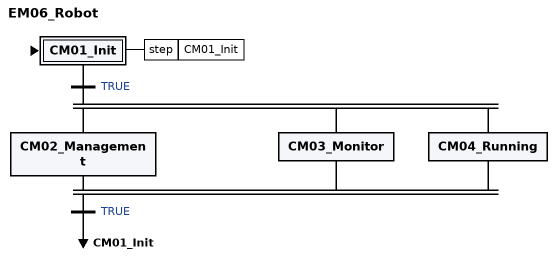
INITIAL_STEP CM01_Init:
    CM01_Init(N);  // step action
END_STEP
TRANSITION FROM CM01_Init TO (CM02_Management, CM03_Monitor, CM04_Running)
    := TRUE;
END_TRANSITION
STEP CM02_Management:
END_STEP
STEP CM03_Monitor:
END_STEP
STEP CM04_Running:
END_STEP
TRANSITION FROM (CM02_Management, CM03_Monitor, CM04_Running) TO CM01_Init
    := TRUE;
END_TRANSITION

ACTION CM01_Init:

END_ACTION

ACTION CM02_Management:
// NETWORK 1
END_ACTION

ACTION CM03_Monitor:
// NETWORK 1
END_ACTION

ACTION CM04_Running:
// NETWORK 1
END_ACTION

END_PROGRAM

// ---- POUs/S03_Robot_1/UN01_StateMachineRobot_1.TcPOU
PROGRAM UN01_StateMachineRobot_1
VAR
	FB_StateMachineInfeed	: FB_StateManager;
	FB_StateMachinePlacing_1: FB_StateManager;
	FB_StateMachinePlacing_2: FB_StateManager;
	FB_StateMachinePlacing_3: FB_StateManager;
	FB_StateMachinePlacing_4: FB_StateManager;
	FB_StateMachineRobot	: FB_StateManager;
END_VAR

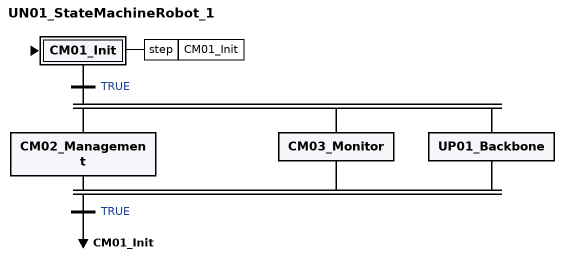
INITIAL_STEP CM01_Init:
    CM01_Init(N);  // step action
END_STEP
TRANSITION FROM CM01_Init TO (CM02_Management, CM03_Monitor, UP01_Backbone)
    := TRUE;
END_TRANSITION
STEP CM02_Management:
END_STEP
STEP CM03_Monitor:
END_STEP
STEP UP01_Backbone:
END_STEP
TRANSITION FROM (CM02_Management, CM03_Monitor, UP01_Backbone) TO CM01_Init
    := TRUE;
END_TRANSITION

ACTION CM01_Init:
//Infeed
Data_GVL.bFL_StartInfeed 			:= Data_GVL.bStartButton OR HMI_GVL.bStartButtonInfeed;
Data_GVL.bFL_StopInfeed 			:= Data_GVL.bStopButton OR HMI_GVL.bStopButtonInfeed;
Data_GVL.bFL_ResetInfeed 			:= Data_GVL.bResetButton OR HMI_GVL.bResetButtonInfeed;
Data_GVL.bFL_AutoManuaModeInfeed 	:= NOT Data_GVL.StateMachineInfeed.Running AND HMI_GVL.bTestModeEnableInfeed;
//Placing 1
Data_GVL.bFL_StartPlacing_1 		:= Data_GVL.bStartButton OR HMI_GVL.bStartButtonPlacing_1;
Data_GVL.bFL_StopPlacing_1 			:= Data_GVL.bStopButton OR HMI_GVL.bStopButtonPlacing_1;
Data_GVL.bFL_ResetPlacing_1			:= Data_GVL.bResetButton OR HMI_GVL.bResetButtonPlacing_1;
Data_GVL.bFL_AutoManuaModePlacing_1 := NOT Data_GVL.StateMachinePlacing_1.Running AND HMI_GVL.bTestModeEnablePlacing_1;
//Placing 2
Data_GVL.bFL_StartPlacing_2 		:= Data_GVL.bStartButton OR HMI_GVL.bStartButtonPlacing_2;
Data_GVL.bFL_StopPlacing_2 			:= Data_GVL.bStopButton OR HMI_GVL.bStopButtonPlacing_2;
Data_GVL.bFL_ResetPlacing_2			:= Data_GVL.bResetButton OR HMI_GVL.bResetButtonPlacing_2;
Data_GVL.bFL_AutoManuaModePlacing_2 := NOT Data_GVL.StateMachinePlacing_2.Running AND HMI_GVL.bTestModeEnablePlacing_2;
//Placing 3
Data_GVL.bFL_StartPlacing_3 		:= Data_GVL.bStartButton OR HMI_GVL.bStartButtonPlacing_3;
Data_GVL.bFL_StopPlacing_3 			:= Data_GVL.bStopButton OR HMI_GVL.bStopButtonPlacing_3;
Data_GVL.bFL_ResetPlacing_3			:= Data_GVL.bResetButton OR HMI_GVL.bResetButtonPlacing_3;
Data_GVL.bFL_AutoManuaModePlacing_3 := NOT Data_GVL.StateMachinePlacing_3.Running AND HMI_GVL.bTestModeEnablePlacing_3;
//Placing 4
Data_GVL.bFL_StartPlacing_4 		:= Data_GVL.bStartButton OR HMI_GVL.bStartButtonPlacing_4;
Data_GVL.bFL_StopPlacing_4 			:= Data_GVL.bStopButton OR HMI_GVL.bStopButtonPlacing_4;
Data_GVL.bFL_ResetPlacing_4			:= Data_GVL.bResetButton OR HMI_GVL.bResetButtonPlacing_4;
Data_GVL.bFL_AutoManuaModePlacing_4 := NOT Data_GVL.StateMachinePlacing_4.Running AND HMI_GVL.bTestModeEnablePlacing_4;
//Robot
Data_GVL.bFL_StartRobot 			:= Data_GVL.bStartButton OR HMI_GVL.bStartButtonRobot;
Data_GVL.bFL_StopRobot 				:= Data_GVL.bStopButton OR HMI_GVL.bStopButtonRobot;
Data_GVL.bFL_ResetRobot 			:= Data_GVL.bResetButton OR HMI_GVL.bResetButtonRobot;
Data_GVL.bFL_AutoManuaModeRobot 	:= NOT Data_GVL.StateMachineRobot.Running AND HMI_GVL.bTestModeEnableRobot;
END_ACTION

ACTION CM02_Management:
// NETWORK 1
END_ACTION

ACTION CM03_Monitor:
// NETWORK 1
END_ACTION

ACTION UP01_Backbone:
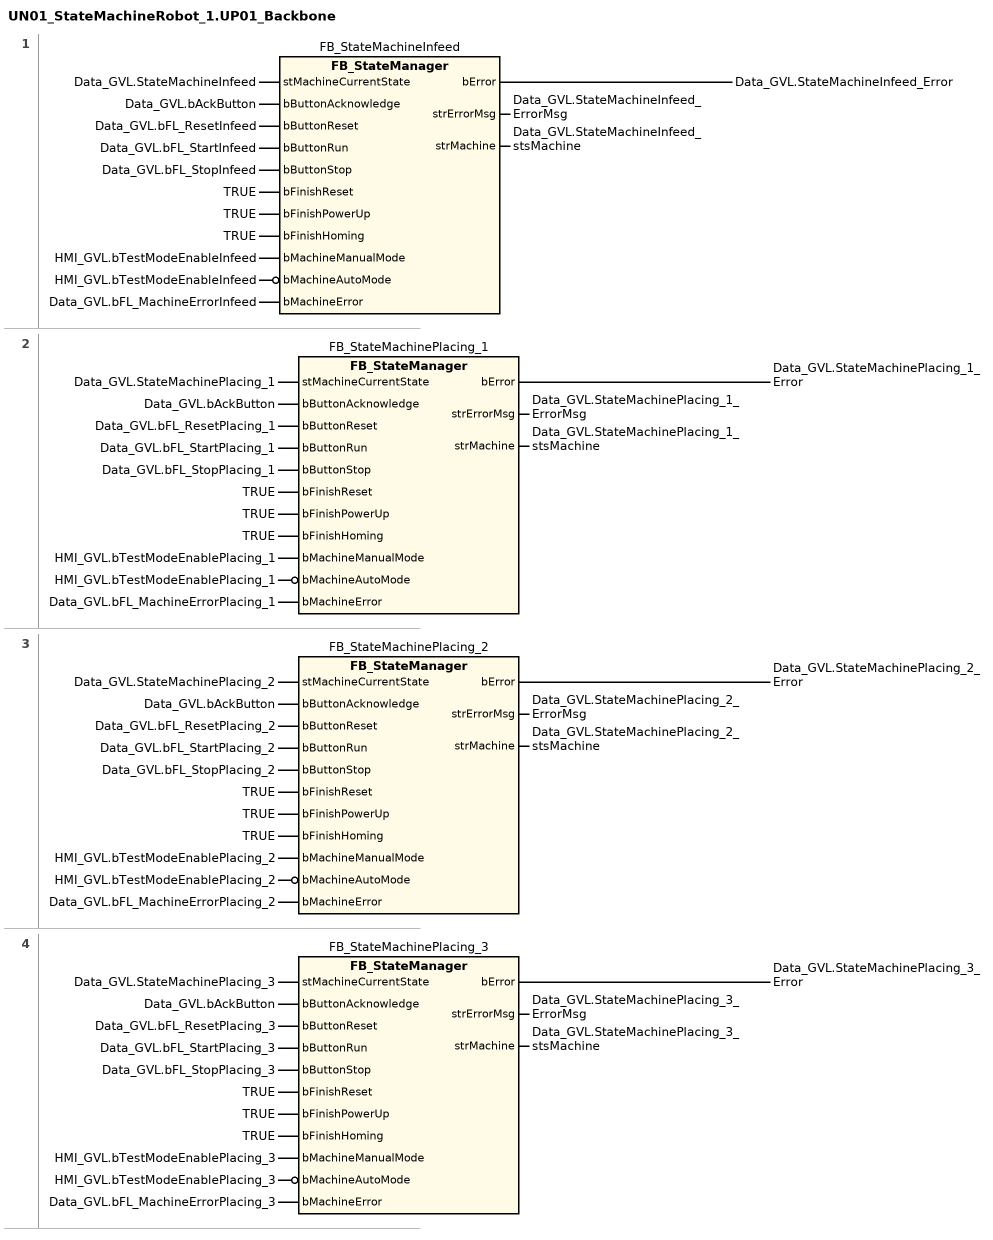
// NETWORK 1
FB_StateMachineInfeed(
    stMachineCurrentState := Data_GVL.StateMachineInfeed,
    bButtonAcknowledge := Data_GVL.bAckButton,
    bButtonReset := Data_GVL.bFL_ResetInfeed,
    bButtonRun := Data_GVL.bFL_StartInfeed,
    bButtonStop := Data_GVL.bFL_StopInfeed,
    bFinishReset := TRUE,
    bFinishPowerUp := TRUE,
    bFinishHoming := TRUE,
    bMachineManualMode := HMI_GVL.bTestModeEnableInfeed,
    bMachineAutoMode := NOT HMI_GVL.bTestModeEnableInfeed,
    bMachineError := Data_GVL.bFL_MachineErrorInfeed,
    strErrorMsg => Data_GVL.StateMachineInfeed_ErrorMsg,
    strMachine => Data_GVL.StateMachineInfeed_stsMachine); // FB_StateManager
Data_GVL.StateMachineInfeed_Error := FB_StateMachineInfeed.bError;

// NETWORK 2
FB_StateMachinePlacing_1(
    stMachineCurrentState := Data_GVL.StateMachinePlacing_1,
    bButtonAcknowledge := Data_GVL.bAckButton,
    bButtonReset := Data_GVL.bFL_ResetPlacing_1,
    bButtonRun := Data_GVL.bFL_StartPlacing_1,
    bButtonStop := Data_GVL.bFL_StopPlacing_1,
    bFinishReset := TRUE,
    bFinishPowerUp := TRUE,
    bFinishHoming := TRUE,
    bMachineManualMode := HMI_GVL.bTestModeEnablePlacing_1,
    bMachineAutoMode := NOT HMI_GVL.bTestModeEnablePlacing_1,
    bMachineError := Data_GVL.bFL_MachineErrorPlacing_1,
    strErrorMsg => Data_GVL.StateMachinePlacing_1_ErrorMsg,
    strMachine => Data_GVL.StateMachinePlacing_1_stsMachine); // FB_StateManager
Data_GVL.StateMachinePlacing_1_Error := FB_StateMachinePlacing_1.bError;

// NETWORK 3
FB_StateMachinePlacing_2(
    stMachineCurrentState := Data_GVL.StateMachinePlacing_2,
    bButtonAcknowledge := Data_GVL.bAckButton,
    bButtonReset := Data_GVL.bFL_ResetPlacing_2,
    bButtonRun := Data_GVL.bFL_StartPlacing_2,
    bButtonStop := Data_GVL.bFL_StopPlacing_2,
    bFinishReset := TRUE,
    bFinishPowerUp := TRUE,
    bFinishHoming := TRUE,
    bMachineManualMode := HMI_GVL.bTestModeEnablePlacing_2,
    bMachineAutoMode := NOT HMI_GVL.bTestModeEnablePlacing_2,
    bMachineError := Data_GVL.bFL_MachineErrorPlacing_2,
    strErrorMsg => Data_GVL.StateMachinePlacing_2_ErrorMsg,
    strMachine => Data_GVL.StateMachinePlacing_2_stsMachine); // FB_StateManager
Data_GVL.StateMachinePlacing_2_Error := FB_StateMachinePlacing_2.bError;

// NETWORK 4
FB_StateMachinePlacing_3(
    stMachineCurrentState := Data_GVL.StateMachinePlacing_3,
    bButtonAcknowledge := Data_GVL.bAckButton,
    bButtonReset := Data_GVL.bFL_ResetPlacing_3,
    bButtonRun := Data_GVL.bFL_StartPlacing_3,
    bButtonStop := Data_GVL.bFL_StopPlacing_3,
    bFinishReset := TRUE,
    bFinishPowerUp := TRUE,
    bFinishHoming := TRUE,
    bMachineManualMode := HMI_GVL.bTestModeEnablePlacing_3,
    bMachineAutoMode := NOT HMI_GVL.bTestModeEnablePlacing_3,
    bMachineError := Data_GVL.bFL_MachineErrorPlacing_3,
    strErrorMsg => Data_GVL.StateMachinePlacing_3_ErrorMsg,
    strMachine => Data_GVL.StateMachinePlacing_3_stsMachine); // FB_StateManager
Data_GVL.StateMachinePlacing_3_Error := FB_StateMachinePlacing_3.bError;

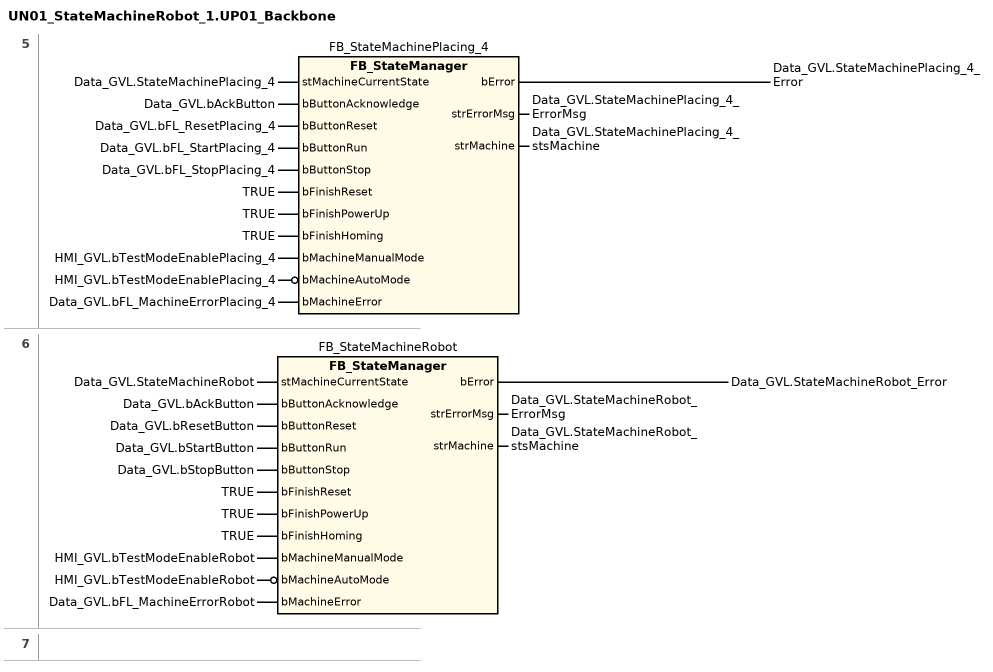
// NETWORK 5
FB_StateMachinePlacing_4(
    stMachineCurrentState := Data_GVL.StateMachinePlacing_4,
    bButtonAcknowledge := Data_GVL.bAckButton,
    bButtonReset := Data_GVL.bFL_ResetPlacing_4,
    bButtonRun := Data_GVL.bFL_StartPlacing_4,
    bButtonStop := Data_GVL.bFL_StopPlacing_4,
    bFinishReset := TRUE,
    bFinishPowerUp := TRUE,
    bFinishHoming := TRUE,
    bMachineManualMode := HMI_GVL.bTestModeEnablePlacing_4,
    bMachineAutoMode := NOT HMI_GVL.bTestModeEnablePlacing_4,
    bMachineError := Data_GVL.bFL_MachineErrorPlacing_4,
    strErrorMsg => Data_GVL.StateMachinePlacing_4_ErrorMsg,
    strMachine => Data_GVL.StateMachinePlacing_4_stsMachine); // FB_StateManager
Data_GVL.StateMachinePlacing_4_Error := FB_StateMachinePlacing_4.bError;

// NETWORK 6
FB_StateMachineRobot(
    stMachineCurrentState := Data_GVL.StateMachineRobot,
    bButtonAcknowledge := Data_GVL.bAckButton,
    bButtonReset := Data_GVL.bResetButton,
    bButtonRun := Data_GVL.bStartButton,
    bButtonStop := Data_GVL.bStopButton,
    bFinishReset := TRUE,
    bFinishPowerUp := TRUE,
    bFinishHoming := TRUE,
    bMachineManualMode := HMI_GVL.bTestModeEnableRobot,
    bMachineAutoMode := NOT HMI_GVL.bTestModeEnableRobot,
    bMachineError := Data_GVL.bFL_MachineErrorRobot,
    strErrorMsg => Data_GVL.StateMachineRobot_ErrorMsg,
    strMachine => Data_GVL.StateMachineRobot_stsMachine); // FB_StateManager
Data_GVL.StateMachineRobot_Error := FB_StateMachineRobot.bError;

// NETWORK 7
END_ACTION

END_PROGRAM

// ---- POUs/Functions Blocks/BLINK.TcPOU
FUNCTION_BLOCK BLINK
VAR_INPUT
	F_Enable: BOOL;
	TimeHigh: TIME:=T#1S;
	TimeLow: TIME:=T#1s;
END_VAR
VAR_OUTPUT
	Output: BOOL;
END_VAR
VAR
	SeqIndex: INT;
	Timer: TON;
END_VAR

IF F_Enable THEN
	CASE SeqIndex OF
		0:
			Output:=TRUE;
			Timer(IN:=TRUE,PT:=TimeHigh);
			IF Timer.Q THEN
				Timer(IN:=FALSE);
				SeqIndex:=10;
			END_IF
		10:
			Output:=FALSE;
			Timer(IN:=TRUE,PT:=TimeLow);
			IF Timer.Q THEN
				Timer(IN:=FALSE);
				SeqIndex:=0;
			END_IF
	END_CASE
ELSE
	SeqIndex:=0;
	Timer(IN:=FALSE);
	Output:=FALSE;
END_IF

END_FUNCTION_BLOCK

// ---- POUs/Functions Blocks/Pneumatic_2Coil_Management.TcPOU
FUNCTION_BLOCK Pneumatic_2Coil_Management //V1.0
// Function block untuk mengolah faceplate dan watchdog pneumatic valve 2 coil
//	UDT dependencies:
	(*  
	1. stPneumatic2 v1.0 	*)

//	Changelog:
	(* 
	
	v1.0 [27.12.2021] Start development function block - Fabrilian Asali	*)	

VAR_INPUT
	bEnable						: BOOL;		
	bTriggerPneumaticRetract	: BOOL;
	bTriggerPneumaticAdvanced	: BOOL;
	bTriggerBoth				: BOOL;
	bReleaseBoth				: BOOL;
	bTestMode					: BOOL;
	bResetError					: BOOL;
	bBypassSensorRetract		: BOOL;
	bBypassSensorAdvanced		: BOOL;
	bBypassPreCheckSensor		: BOOL;
	xIn_SensorRetract			: BOOL;
	xIn_SensorAdvanced			: BOOL;
	TimerWatchdogRetract		: TIME := T#5S;
	TimerWatchdogAdvanced		: TIME := T#5S;
	TimerWatchdogPreRetract		: TIME := T#5S;
	TimerWatchdogPreAdvanced	: TIME := T#5S;
	TimerValve					: TIME := T#25MS;
END_VAR

VAR_OUTPUT
	bError						: BOOL;
	ErrorID						: INT;
	ErrorMsg					: STRING;
END_VAR

VAR_IN_OUT
	Pneumatic			: stPneumatic2;
END_VAR

VAR
	SeqIndex					: INT;
	InitSeqIndex				: INT;
	WatchdogTimer				: TON;
	ValveTimer					: TON;
	bInit						: BOOL;
END_VAR
VAR // added by the converter: edge detectors and wires of the graphical bodies
    _w1 : BOOL;
    _rt1, _rt2, _rt3, _rt4 : R_TRIG;
END_VAR

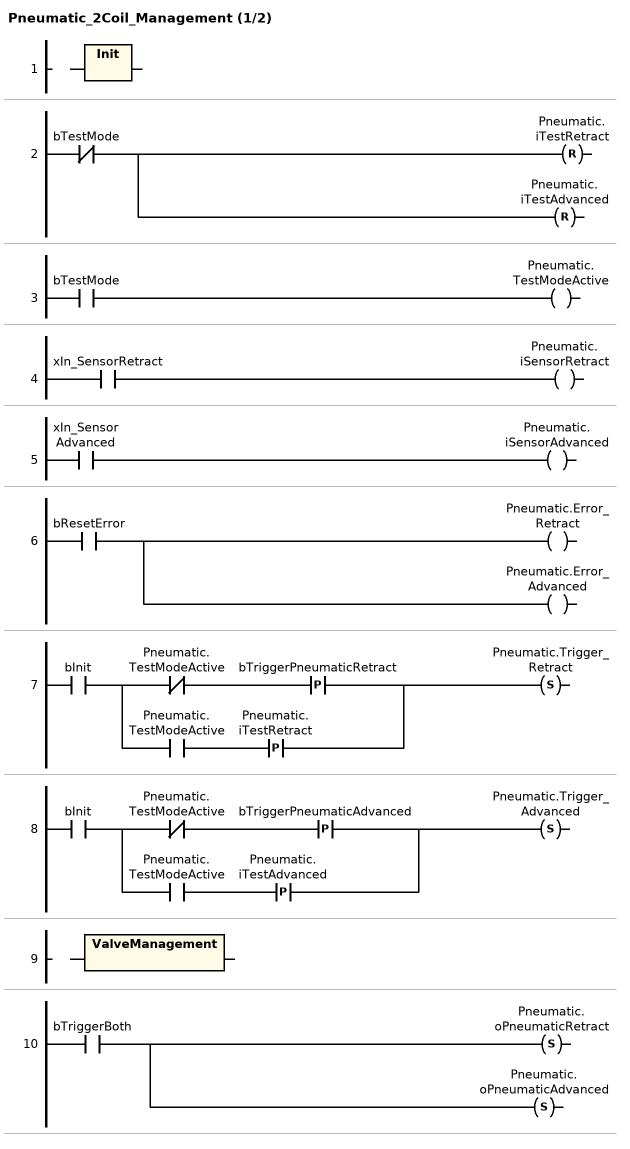
// NETWORK 1
Init();

// NETWORK 2
_w1 := NOT bTestMode;
Pneumatic.iTestRetract R= _w1;
Pneumatic.iTestAdvanced R= _w1;

// NETWORK 3
Pneumatic.TestModeActive := bTestMode;

// NETWORK 4
Pneumatic.iSensorRetract := xIn_SensorRetract;

// NETWORK 5
Pneumatic.iSensorAdvanced := xIn_SensorAdvanced;

// NETWORK 6
Pneumatic.Error_Retract := bResetError;
Pneumatic.Error_Advanced := bResetError;

// NETWORK 7
_rt1(CLK := bTriggerPneumaticRetract);
_rt2(CLK := Pneumatic.iTestRetract);
Pneumatic.Trigger_Retract S= bInit AND (NOT Pneumatic.TestModeActive AND _rt1.Q OR Pneumatic.TestModeActive AND _rt2.Q);

// NETWORK 8
_rt3(CLK := bTriggerPneumaticAdvanced);
_rt4(CLK := Pneumatic.iTestAdvanced);
Pneumatic.Trigger_Advanced S= bInit AND (NOT Pneumatic.TestModeActive AND _rt3.Q OR Pneumatic.TestModeActive AND _rt4.Q);

// NETWORK 9
ValveManagement();

// NETWORK 10
Pneumatic.oPneumaticRetract S= bTriggerBoth;
Pneumatic.oPneumaticAdvanced S= bTriggerBoth;

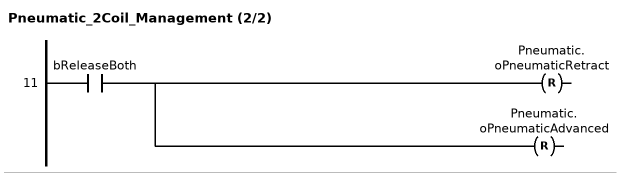
// NETWORK 11
Pneumatic.oPneumaticRetract R= bReleaseBoth;
Pneumatic.oPneumaticAdvanced R= bReleaseBoth;

ACTION Init:
IF bResetError THEN
	bError			:= FALSE;
	InitSeqIndex	:= 0;
END_IF


IF bEnable AND NOT bInit THEN
	CASE InitSeqIndex OF
		0:
			IF xIn_SensorRetract THEN
				InitSeqIndex	:= 100;
			ELSIF xin_SensorAdvanced THEN
				InitSeqIndex	:= 200;
			ELSIF NOT xIn_SensorRetract AND NOT xIn_SensorAdvanced THEN
				InitSeqIndex	:= 300;
			ELSE
				ErrorID			:= 1;
				ErrorMsg		:= 'Both Sensor on at Init';
				InitSeqIndex	:= 999;
			END_IF
	
		100:
			Pneumatic.oPneumaticRetract 	:= TRUE;
			InitSeqIndex	:= 1000;
		
		200:
			Pneumatic.oPneumaticAdvanced	:= TRUE;
			InitSeqIndex	:= 1000;
		
		300:
			Pneumatic.oPneumaticRetract		:= TRUE;
			Pneumatic.oPneumaticAdvanced	:= TRUE;
			WatchdogTimer(In:= TRUE, PT:= T#10S);
			IF xIn_SensorRetract THEN
				Pneumatic.oPneumaticAdvanced	:= FALSE;
				InitSeqIndex	:= 1000;
			ELSIF xIn_SensorAdvanced THEN
				Pneumatic.oPneumaticRetract		:= FALSE;
				InitSeqIndex	:= 1000;
			ELSIF WatchdogTimer.Q THEN
				ErrorID			:= 2;
				ErrorMsg		:= 'Pneu Init Failed';
				InitSeqIndex	:= 999;
			END_IF
			
		
		999:
			bError	:= TRUE;
		
		1000:
			bInit	:= TRUE;
		
	END_CASE
END_IF
END_ACTION

ACTION ValveManagement:

IF bResetError THEN
	bError		:= FALSE;
	ErrorID		:= 0;
	ErrorMsg	:= '';
	SeqIndex	:= 0;
END_IF

IF bEnable AND bInit AND NOT bError THEN
	CASE SeqIndex OF
		0:
			IF Pneumatic.Trigger_Retract THEN
				SeqIndex	:= 100;
			ELSIF Pneumatic.Trigger_Advanced THEN
				SeqIndex	:= 200;
			END_IF
			
		100:
			Pneumatic.Trigger_Retract	:= FALSE;
			IF NOT bBypassPreCheckSensor THEN
				WatchdogTimer(In:= TRUE, PT:= TimerWatchdogPreRetract);
				IF Pneumatic.iSensorAdvanced THEN
					WatchdogTimer(In:= FALSE);
					SeqIndex	:= 105;
				ELSIF WatchdogTimer.Q THEN
					WatchdogTimer(In:= FALSE);
					Pneumatic.Error_Retract := TRUE;
					ErrorID					:= 10;
					ErrorMsg				:= 'Error PreCheck Retract';
					SeqIndex	:= 999;
				END_IF
			ELSE
				SeqIndex	:= 105;
			END_IF
	
		105:	
			Pneumatic.oPneumaticRetract		:= TRUE;
			Pneumatic.oPneumaticAdvanced	:= TRUE;
			ValveTimer(In:= TRUE, PT:= TimerValve);
			IF ValveTimer.Q THEN
				ValveTimer(In:= FALSE);
				Pneumatic.oPneumaticAdvanced	:= FALSE;
				SeqIndex	:= 110;
			END_IF
			
		110:
			IF NOT bBypassSensorRetract THEN
				WatchdogTimer(In:= TRUE, PT:= TimerWatchdogRetract);
				IF Pneumatic.iSensorRetract THEN
					WatchdogTimer(In:= FALSE);
					SeqIndex	:= 0;
				ELSIF WatchdogTimer.Q THEN
					WatchdogTimer(In:= FALSE);
					Pneumatic.Error_Retract := TRUE;
					ErrorID					:= 11;
					ErrorMsg				:= 'Error Watchdog Retract';
				END_IF
			ELSE
				SeqIndex	:= 0;
			END_IF
		
			
		200:
			Pneumatic.Trigger_Advanced	:= FALSE;
			IF NOT bBypassPreCheckSensor THEN
				WatchdogTimer(In:= TRUE, PT:= TimerWatchdogPreAdvanced);
				IF Pneumatic.iSensorRetract THEN
					WatchdogTimer(In:= FALSE);
					SeqIndex	:= 210;
				ELSIF WatchdogTimer.Q THEN
					WatchdogTimer(In:= FALSE);
					Pneumatic.Error_Advanced := TRUE;
					ErrorID					:= 20;
					ErrorMsg				:= 'Error PreCheck Advanced';
					SeqIndex	:= 999;
				END_IF
			ELSE
				SeqIndex	:= 205;
			END_IF				
		
		205:
			Pneumatic.oPneumaticRetract		:= TRUE;
			Pneumatic.oPneumaticAdvanced	:= TRUE;
			ValveTimer(In:= TRUE, PT:= TimerValve);
			IF ValveTimer.Q THEN
				Pneumatic.oPneumaticRetract	:= FALSE;
				SeqIndex	:= 210;
			END_IF	
			
		210:
			IF NOT bBypassSensorAdvanced THEN
				WatchdogTimer(In:= TRUE, PT:= TimerWatchdogAdvanced);
				IF Pneumatic.iSensorAdvanced THEN
					WatchdogTimer(In:= FALSE);
					SeqIndex	:= 0;
				ELSIF WatchdogTimer.Q THEN
					WatchdogTimer(In:= FALSE);
					Pneumatic.Error_Advanced := TRUE;
					ErrorID					:= 21;
					ErrorMsg				:= 'Error Watchdog Advanced';
				END_IF
			ELSE
				SeqIndex	:= 0;
			END_IF					
	
		999:
			bError	:= TRUE;	
	
	
	END_CASE
	
ELSE
	SeqIndex	:= 0;
	WatchdogTimer(IN:= FALSE);
END_IF
END_ACTION

END_FUNCTION_BLOCK
